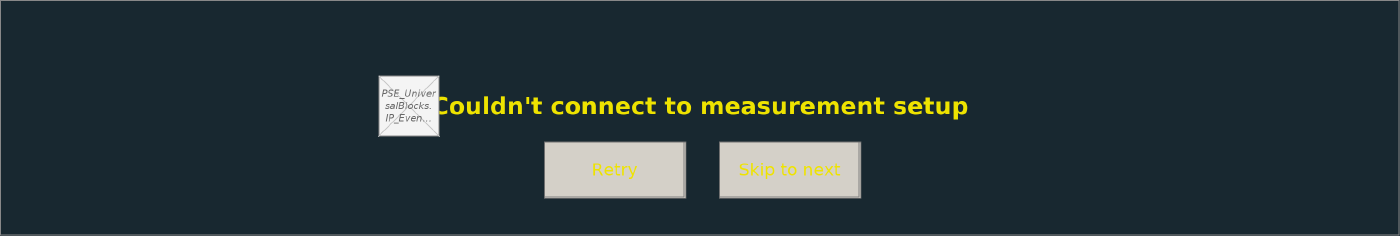
VISUALIZATION InitializingFixtureConnectionFailed  // 1480x250
VAR_IN_OUT
	btnFixtureConnectionRetry	: BOOL;
	btnFixtureConnectionSkip	: BOOL;
END_VAR
    Label (0,92 1480x40), "Couldn't connect to measurement setup"
    Button (575,150 150x60), "Retry"
        toggle btnFixtureConnectionRetry
    Button (760,150 150x60), "Skip to next"
        toggle btnFixtureConnectionSkip
    Image (400,80 64x64), image: PSE_UniversalBlocks.IP_EventSeverity.warning
END_VISUALIZATION

(* stored: Version 1.1.0.1, ProductVersion 3.1.4024.9
   Visu InitializingFixtureConnectionFailed: Id {c9812c56-0892-4340-809c-affabf346e6a} *)
